Fanuc KAREL source: kb00121.KL

-- PROVISIONAL review KL for V770-1; original PC SHA256 c21a68400256553e934b276ba3919fdacc46634075e7401a31d8ce6852c39099
-- Incomplete behavior may be omitted. Consult companion uncertainty JSON. Do not deploy.
PROGRAM KB00121
%NOLOCKGROUP
BEGIN
  -- UNRESOLVED_PC offsets 5-12; opcodes 9D,23
  -- UNRESOLVED_PC offsets 17-24; opcodes 9D,23
  -- UNRESOLVED_PC offsets 29-39; opcodes 9D,22,9D,33,35
  -- UNRESOLVED_PC offsets 44-51; opcodes 9D,23
  -- UNRESOLVED_PC offsets 56-90; opcodes 27,22,22,22,22,22,31
  -- UNRESOLVED_PC offsets 95-99; opcodes 7F
END KB00121
